// Mitsubishi GX Works2 project: 시퀀스 무한반복 예제2 (답안)   PLC: Q03UDV

PROGRAM MAIN
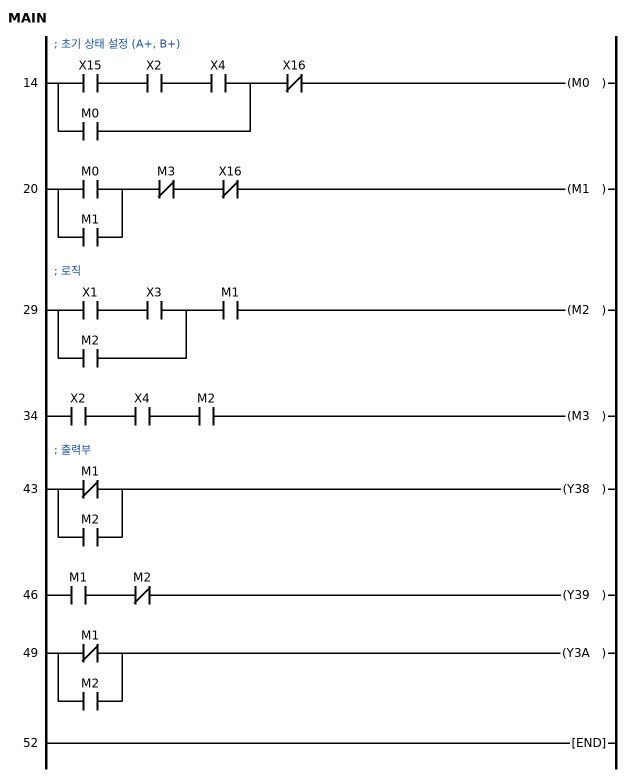
; 초기 상태 설정 (A+, B+)
14    LD      X15
      AND     X2
      AND     X4
      OR      M0
      ANI     X16
      OUT     M0
20    LD      M0
      OR      M1
      ANI     M3
      ANI     X16
      OUT     M1
; 로직
29    LD      X1
      AND     X3
      OR      M2
      AND     M1
      OUT     M2
34    LD      X2
      AND     X4
      AND     M2
      OUT     M3
; 출력부
43    LDI     M1
      OR      M2
      OUT     Y38
46    LD      M1
      ANI     M2
      OUT     Y39
49    LDI     M1
      OR      M2
      OUT     Y3A
52    END
END_PROGRAM
